// TIA Portal V20 export
// export: Created 2025-12-01T14:57:21.9930818Z, ExportSetting None, DisplayName Totally Integrated Automation Portal, DisplayVersion V20 Update 3, DisplayName TIA Portal Openness, DisplayVersion V20 Update 3, DisplayName TIA Portal Version Control Interface, DisplayVersion V20 Update 3, DisplayName STEP 7 Professional, DisplayVersion V20 Update 3, DisplayName STEP 7 Safety, DisplayVersion V20 Update 2, DisplayName WinCC Basic/Comfort/Advanced, DisplayVersion V20 Update 3, DisplayName WinCC Professional, DisplayVersion V20 Update 3, DisplayName WinCC Unified, DisplayVersion V20 Update 3
DATA_BLOCK "DB753_PantallaNº04"   // DB753
{ S7_Optimized_Access := 'FALSE' }
AUTHOR : PANTALLA
NAME : 20160415
VERSION : 5.0
// stored: AutoNumber false
   VAR
      HMI { S7_SetPoint := 'True'} : "UDT_HMI";
   END_VAR
BEGIN
END_DATA_BLOCK
